FUNCTION_BLOCK FB_Intersection
VAR
	_phase : E_Phase := E_Phase.AllRed;

    // Concrete instances — these actually own the light objects
    _nsLightImpl : FB_TrafficLight;
    _ewLightImpl : FB_TrafficLight;

    // Interface references — the intersection talks to lights via the contract
    _nsLight : ITrafficLight;
    _ewLight : ITrafficLight;
END_VAR

METHOD PUBLIC Advance
VAR
END_VAR
// Normal-mode behavior for now.
// A control-mode CASE (Emergency, NightFlash, Manual) would wrap this later.
RunNormalCycle();
ApplyPhaseToLights();
END_METHOD

METHOD PRIVATE ApplyPhaseToLights
VAR_INPUT
END_VAR
CASE _phase OF

    E_Phase.AllRed:
        _nsLight.CurrentState := E_LightState.Red;
        _ewLight.CurrentState := E_LightState.Red;

    E_Phase.NorthSouthFlowing:
        _nsLight.CurrentState := E_LightState.Green;
        _ewLight.CurrentState := E_LightState.Red;

    E_Phase.NorthSouthClearing:
        _nsLight.CurrentState := E_LightState.Amber;
        _ewLight.CurrentState := E_LightState.Red;

    E_Phase.EastWestFlowing:
        _nsLight.CurrentState := E_LightState.Red;
        _ewLight.CurrentState := E_LightState.Green;

    E_Phase.EastWestClearing:
        _nsLight.CurrentState := E_LightState.Red;
        _ewLight.CurrentState := E_LightState.Amber;

END_CASE
END_METHOD

PROPERTY CurrentPhase : E_Phase
GET
CurrentPhase := _phase;
END_GET
END_PROPERTY

PROPERTY EastWestState : E_LightState
GET
EastWestState := _ewLight.CurrentState;
END_GET
END_PROPERTY

METHOD FB_init : BOOL
VAR_INPUT
	bInitRetains : BOOL; // if TRUE, the retain variables are initialized (warm start / cold start)
	bInCopyCode : BOOL;  // if TRUE, the instance afterwards gets moved into the copy code (online change)
END_VAR
// Point interface references at the concrete instances (runs once, at creation)
_nsLight := _nsLightImpl;
_ewLight := _ewLightImpl;
END_METHOD

PROPERTY NorthSouthState : E_LightState
GET
NorthSouthState := _nsLight.CurrentState;
END_GET
END_PROPERTY

METHOD PRIVATE RunNormalCycle
VAR
END_VAR
CASE _phase OF

    E_Phase.AllRed:
        _phase := E_Phase.NorthSouthFlowing;

    E_Phase.NorthSouthFlowing:
        _phase := E_Phase.NorthSouthClearing;

    E_Phase.NorthSouthClearing:
        _phase := E_Phase.EastWestFlowing;

    E_Phase.EastWestFlowing:
        _phase := E_Phase.EastWestClearing;

    E_Phase.EastWestClearing:
        _phase := E_Phase.NorthSouthFlowing;  

END_CASE
END_METHOD

END_FUNCTION_BLOCK

(* stored: Version 1.1.0.1, ProductVersion 3.1.4024.12
   POU FB_Intersection: Id {e5cfebb4-1149-4b39-adfb-333fbff08c59}, SpecialFunc None
   Method Advance: Id {bdb8fcda-c6d7-40a4-85ce-59097b5ad1f7}
   Method ApplyPhaseToLights: Id {4ea9a396-25b9-4204-ad57-326c4b63df04}
   Property CurrentPhase: Id {51a0cff2-4575-44fb-abb8-3f8e1e191446}
   Get Get: Id {491615fe-6f28-44e3-a74d-1231442b9920}
   Property EastWestState: Id {eaaaaa52-e805-400d-a3c8-7f085e87c6f9}
   Get Get: Id {9cf8c84d-4971-4fcd-b25b-2b4795173e14}
   Method FB_init: Id {bf28138a-dec2-4334-9ac1-1994ca97fde8}
   Property NorthSouthState: Id {9d6778a6-7c76-4503-876a-525b44455ef7}
   Get Get: Id {0e3b2ca8-1bd4-4186-8d53-48c298ad5621}
   Method RunNormalCycle: Id {49c2bdac-7879-4d9e-8937-f658ecf7a5df} *)
